// TwinCAT 3 PLC project Simulink_Crane
// ProgramVersion: 3.1.4024.0
// libraries:
//   Tc2_Standard, * (Beckhoff Automation GmbH)
//   Tc2_System, * (Beckhoff Automation GmbH)
//   Tc3_Module, * (Beckhoff Automation GmbH)
// project tree:
//   / PlcTask.TcTTO, Simulator.TcTTO
//   POUs/ MAIN.TcPOU, P_Simulator.TcPOU

CONFIGURATION Simulink_Crane
    RESOURCE PLC ON TwinCAT3
        TASK PlcTask(INTERVAL := T#10ms, PRIORITY := 20);
        TASK Simulator(INTERVAL := T#100us, PRIORITY := 1);
        PROGRAM MAIN WITH PlcTask : MAIN;
        PROGRAM P_Simulator WITH Simulator : P_Simulator;
    END_RESOURCE
END_CONFIGURATION

// ---- POUs/MAIN.TcPOU
PROGRAM MAIN
VAR
END_VAR

END_PROGRAM

// ---- POUs/P_Simulator.TcPOU
PROGRAM P_Simulator
VAR
END_VAR

END_PROGRAM
